{attribute 'linkalways'} 
{attribute 'no_explicit_call' := 'This FB is a CLASS and must be accessed using methods or properties'}
{attribute 'enable_dynamic_creation'}
FUNCTION_BLOCK FINAL MIN_DWORD EXTENDS Node
VAR
	in1 : _DWORD(0);
	in2 : _DWORD(0);
	out : _DWORD(0);
END_VAR

METHOD PUBLIC Clone : I_Node
VAR
	pNode : POINTER TO MIN_DWORD;
END_VAR
pNode := __NEW(MIN_DWORD);
Clone := pNode^;
END_METHOD

METHOD FB_init : BOOL
VAR_INPUT
	bInitRetains : BOOL; // if TRUE, the retain variables are initialized (warm start / cold start)
	bInCopyCode : BOOL;  // if TRUE, the instance afterwards gets moved into the copy code (online change)
END_VAR
AddInput('in1',THIS^.in1);
AddInput('in2',THIS^.in2);
AddOutput('out', THIS^.out);
END_METHOD

METHOD PROTECTED OnExecute
VAR
END_VAR
out.Value := MIN(in1.Value, in2.Value);
END_METHOD

END_FUNCTION_BLOCK

(* stored: Version 1.1.0.1, ProductVersion 3.1.4024.15
   POU MIN_DWORD: Id {d1e4fe41-72bb-4e0c-92f0-18b949f360c7}, SpecialFunc None
   Folder Constructor: Id {8e97ef48-9641-4885-a8e1-3b0986673e80}
   Method Clone: Id {de8b3db9-612e-4c5d-b6ae-69d603728ce0}
   Method FB_init: Id {17261159-ae1c-4090-822b-346d9cae8349}
   Method OnExecute: Id {e5236f2a-4671-4cd6-9588-93a7e51dbebb} *)
